(* CoDeSys 2.3.9.35 project: Semaforo3.pro *)
(* Author: Altus *)
(* Libraries: DU35x.lib 7.7.11 15:59:13, Navigation.lib 15.7.11 10:06:00, SysLibTargetVisu.lib 26.11.08 09:53:28, Standard.lib 26.11.08 09:46:20, Iecsfc.lib 26.11.08 09:46:14, SYSLIBCALLBACK.LIB 26.11.08 09:53:30 *)

(* PLC configuration (modules and I/O channels)
Configuração do CP [Root] node -1, in %IB0 out %QB0
  Comunicação [Comunica] node 0, in %IB0 out %QB0
    COM1 [COM1] node 0, in %IB0 out %QB0 {BaudRate = 115200; Paridade = Sem Paridade; StopBits = 1 Stop Bit; Modem = Sem RTS/CTS; Delay = 5}
      MToolIEC [Codesys] node 0, in %IB0 out %QB0
    COM2 [COM2] node 1, in %IB0 out %QB0 {BaudRate = 115200; Paridade = Sem Paridade; StopBits = 1 Stop Bit; Modem = Sem RTS/CTS; Delay = 5}
      Desabilitada [Desabilitado485] node 0, in %IB0 out %QB0
  Barramento [Barramento] node 1, in %IB0 out %QB0
    Entradas [Entradas] node 0, in %IB0 out %QB0
      Entradas Digitais 0 [Entradas0] node 0, in %IW0 out %QB0
        I00 AT %IX0.0 [BitInput] I0.0
        I01 AT %IX0.1 [BitInput] I0.1
        I02 AT %IX0.2 [BitInput] I0.2
        I03 AT %IX0.3 [BitInput] I0.3
        I04 AT %IX0.4 [BitInput] I0.4
        I05 AT %IX0.5 [BitInput] I0.5
        I06 AT %IX0.6 [BitInput] I0.6
        I07 AT %IX0.7 [BitInput] I0.7
        I08 AT %IX0.8 [BitInput] I0.8
      Entradas Digitais 1 [Entradas1] node 0, in %IW1 out %QB0
        I10 AT %IX1.0 [BitInput] I1.0
        I11 AT %IX1.1 [BitInput] I1.1
        I12 AT %IX1.2 [BitInput] I1.2
        I13 AT %IX1.3 [BitInput] I1.3
        I14 AT %IX1.4 [BitInput] I1.4
        I15 AT %IX1.5 [BitInput] I1.5
        I16 AT %IX1.6 [BitInput] I1.6
        I17 AT %IX1.7 [BitInput] I1.7
        I18 AT %IX1.8 [BitInput] I1.8
      Entradas Digitais 2 [Entradas2] node 0, in %IW2 out %QB0
        I20 AT %IX2.0 [BitInput] I2.0
        I21 AT %IX2.1 [BitInput] I2.1
      Entradas Analógicas [EntradaAnalogica] node 0, in %IW4 out %QB0
        AI0 AT %IW4 [WordInput] AI0 {TipoAnalogica = Channel Disable; FiltroAnalogica = Filter 0 - AI=2ms  / AV=90ms; FundoEscala = 0}
        AI1 AT %IW5 [WordInput] AI1 {TipoAnalogica = Channel Disable; FiltroAnalogica = Filter 0 - AI=2ms  / AV=90ms; FundoEscala = 0}
        AI2 AT %IW6 [WordInput] AI2 {TipoAnalogica = Channel Disable; FiltroAnalogica = Filter 0 - AI=2ms  / AV=90ms; FundoEscala = 0}
        AI3 AT %IW7 [WordInput] AI3 {TipoAnalogica = Channel Disable; FiltroAnalogica = Filter 0 - AI=2ms  / AV=90ms; FundoEscala = 0}
      Entradas Rápidas [EntradasRapidas] node 1, in %IB16 out %QB0
        Bloco 0 [Bloco0] node 0, in %IB16 out %QB0
          Desabilitado [DesabilitadoBloco0] node 0, in %IB16 out %QB0
        Bloco 1 [Bloco1] node 1, in %IB16 out %QB0
          Desabilitado [DesabilitadoBloco1] node 0, in %IB16 out %QB0
        Entrada Configuravél Bloco 0 [EntradaConfiBloco0] node 2, in %IB16 out %QB0
          Contador 0 [EntradaConfContador0] node 0, in %IB16 out %QB0 {EntradaConfiguravelContador = Disable}
        Entrada Configuravél Bloco 1 [EntradaConfiBloco1] node 3, in %IB16 out %QB0
          Contador 2 [EntradaConfContador2] node 0, in %IB16 out %QB0 {EntradaConfiguravelContador = Disable}
    Saídas [Saidas] node 1, in %IB13 out %QB0
      Saídas Digitais 0 [Saidas0] node 0, in %IW0 out %QW0
        Q00 AT %QX0.0 [BitOutput] Q0.0
        Q01 AT %QX0.1 [BitOutput] Q0.1
        Q02 AT %QX0.2 [BitOutput] Q0.2
        Q03 AT %QX0.3 [BitOutput] Q0.3
        Q04 AT %QX0.4 [BitOutput] Q0.4
        Q05 AT %QX0.5 [BitOutput] Q0.5
        Q06 AT %QX0.6 [BitOutput] Q0.6
        Q07 AT %QX0.7 [BitOutput] Q0.7
      Saídas Digitais 1 [Saidas1] node 0, in %IW0 out %QW1
        Q10 AT %QX1.0 [BitOutput] Q1.0
        Q11 AT %QX1.1 [BitOutput] Q1.1
        Q12 AT %QX1.2 [BitOutput] Q1.2
        Q13 AT %QX1.3 [BitOutput] Q1.3
        Q14 AT %QX1.4 [BitOutput] Q1.4
        Q15 AT %QX1.5 [BitOutput] Q1.5
        Q16 AT %QX1.6 [BitOutput] Q1.6
        Q17 AT %QX1.7 [BitOutput] Q1.7
      Saídas Analógicas [SaidaAnalogica] node 0, in %IW0 out %QW3
        AO0 AT %QW3 [WordOutput] AO0 {TipoAnalogica = Channel Disable; FundoEscala = 0}
        AO1 AT %QW4 [WordOutput] AO1 {TipoAnalogica = Channel Disable; FundoEscala = 0}
      Saídas Rápidas [SaidasRapidas] node 1, in %IB0 out %QB10
        Saída Rápida 0 Desabilitada [DesabilitadoF0] node 0, in %IB0 out %QB10
        Saída Rápida 1 Desabilitada [DesabilitadoF1] node 1, in %IB0 out %QB10
      Saídas Comum de Contador [SaidasContador] node 2, in %IB0 out %QB10
        Saída do Bloco 0 Desabilitada [DesabilitadoSaidaBloco0] node 0, in %IB0 out %QB10
        Saída do Bloco 1 Desabilitada [DesabilitadoSaidaBloco1] node 1, in %IB0 out %QB10
  Eventos Externos [Eventos] node 2, in %IB13 out %QB6
    Evento Temporizado [TimerEvent] node 0, in %IB13 out %QB6 {Intervalo = 10}
*)

(* Task configuration *)
TASK PRINCIPAL (PRIORITY := 1, INTERVAL := T#1ms);
	PLC_PRG();
END_TASK
TASK NAVIGATION (PRIORITY := 1, INTERVAL := T#20ms);
	NAVEGA();
END_TASK
TASK VISUALIZATION (PRIORITY := 1, INTERVAL := T#500ms);
	MAINTARGETVISU_PAINT_CODE
END_TASK
TASK KEYBOARD_USAGE (PRIORITY := 1, INTERVAL := T#20ms);
	MAINTARGETVISU_INPUT_CODE
END_TASK

(* POU PLC_PRG, LD *)
PROGRAM PLC_PRG

VAR_INPUT
	Ligar AT %IX0.0: BOOL;
	Problema AT %IX0.1: BOOL;
END_VAR
VAR_OUTPUT
	Vermelho AT %QX1.0: BOOL;
	Vermelho2 AT %QX1.1: BOOL;
	Vermelho3 AT %QX1.2: BOOL;
	Vermelho4 AT %QX1.3: BOOL;
	Vermelho5 AT %QX1.4: BOOL;
	Vermelho6 AT %QX1.5: BOOL;
	Verde AT %QX1.7: BOOL;
	Amarelo AT %QX1.6: BOOL;
	Restart: BOOL;
	Pisca: BOOL;
	Vermelhoteste: BOOL;
	VerdeDois: BOOL;
	VermelhoDois: BOOL;
	AmareloDois: BOOL;
END_VAR
VAR
	T1: TON;
	T2: TON;
	T3: TON;
	T4: TON;
	T5: TON;
	T6: TON;
	T7: TON;
	T8: TON;
	Entrada1: INT;
	Tempo_Vermelho: TIME:= T#90s;
	Entrada2: INT;
	Tempo_Amarelo: TIME:= T#4s;
	Entrada3: INT;
	Tempo_Verde: TIME:= T#55s;
	T9: TON;
	Restart2: BOOL;
	T10: TON;
	T11: TON;
END_VAR
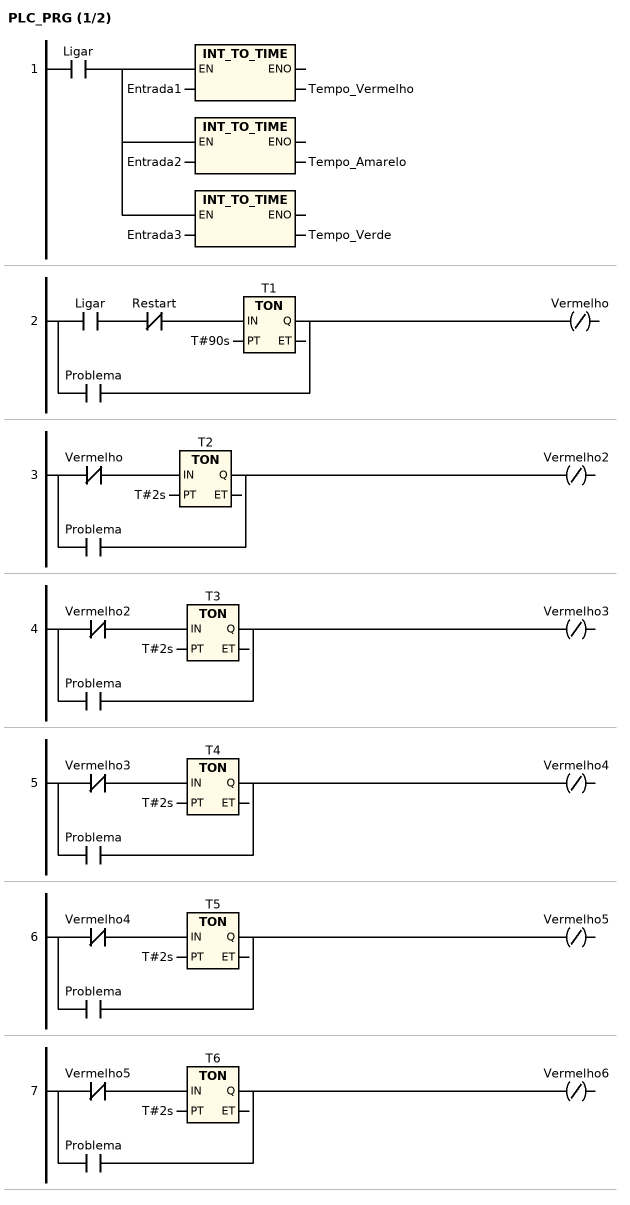
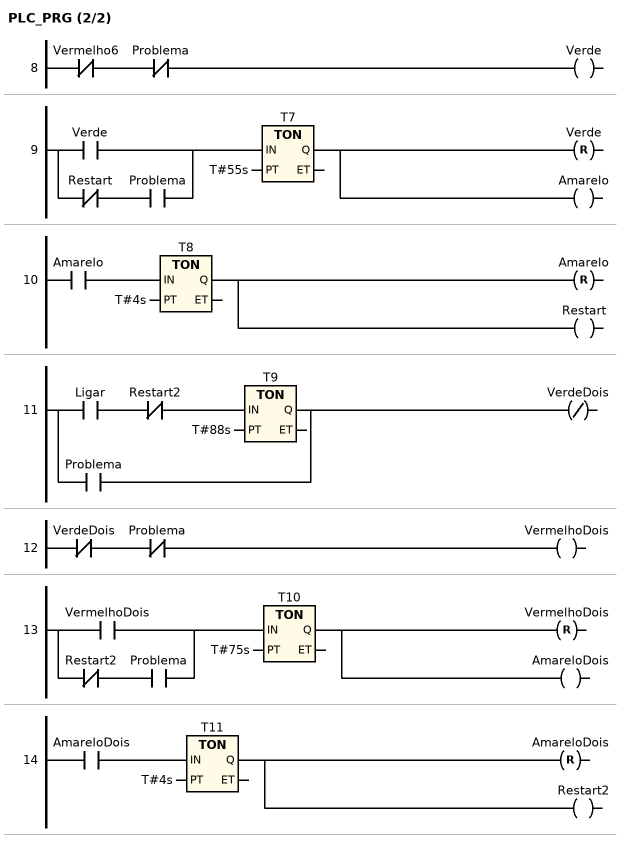
_LD_ (* Ladder Diagram *)
NETWORK 1
	[Ligar]
		EN --- INT_TO_TIME(Entrada1) => Tempo_Vermelho
		EN --- INT_TO_TIME(Entrada2) => Tempo_Amarelo
		EN --- INT_TO_TIME(Entrada3) => Tempo_Verde
NETWORK 2
	{ [Ligar] - [/Restart] - T1:TON(IN: *, PT: T#90s) | [Problema] } --- (/Vermelho)
NETWORK 3
	{ [/Vermelho] - T2:TON(IN: *, PT: T#2s) | [Problema] } --- (/Vermelho2)
NETWORK 4
	{ [/Vermelho2] - T3:TON(IN: *, PT: T#2s) | [Problema] } --- (/Vermelho3)
NETWORK 5
	{ [/Vermelho3] - T4:TON(IN: *, PT: T#2s) | [Problema] } --- (/Vermelho4)
NETWORK 6
	{ [/Vermelho4] - T5:TON(IN: *, PT: T#2s) | [Problema] } --- (/Vermelho5)
NETWORK 7
	{ [/Vermelho5] - T6:TON(IN: *, PT: T#2s) | [Problema] } --- (/Vermelho6)
NETWORK 8
	[/Vermelho6] - [/Problema] --- (Verde)
NETWORK 9
	{ [Verde] | [/Restart] - [Problema] } - T7:TON(IN: *, PT: T#55s) --- (R Verde) (Amarelo)
NETWORK 10
	[Amarelo] - T8:TON(IN: *, PT: T#4s) --- (R Amarelo) (Restart)
NETWORK 11
	{ [Ligar] - [/Restart2] - T9:TON(IN: *, PT: T#88s) | [Problema] } --- (/VerdeDois)
NETWORK 12
	[/VerdeDois] - [/Problema] --- (VermelhoDois)
NETWORK 13
	{ [VermelhoDois] | [/Restart2] - [Problema] } - T10:TON(IN: *, PT: T#75s) --- (R VermelhoDois) (AmareloDois)
NETWORK 14
	[AmareloDois] - T11:TON(IN: *, PT: T#4s) --- (R AmareloDois) (Restart2)
_END_LD_
(* the same logic as Structured Text *)
(* Network 1 *)
IF Ligar THEN
	Tempo_Vermelho := INT_TO_TIME(Entrada1);
	Tempo_Amarelo := INT_TO_TIME(Entrada2);
	Tempo_Verde := INT_TO_TIME(Entrada3);
END_IF;
(* Network 2 *)
T1(IN := Ligar AND NOT Restart, PT := T#90s);
Vermelho := NOT (T1.Q OR Problema);
(* Network 3 *)
T2(IN := NOT Vermelho, PT := T#2s);
Vermelho2 := NOT (T2.Q OR Problema);
(* Network 4 *)
T3(IN := NOT Vermelho2, PT := T#2s);
Vermelho3 := NOT (T3.Q OR Problema);
(* Network 5 *)
T4(IN := NOT Vermelho3, PT := T#2s);
Vermelho4 := NOT (T4.Q OR Problema);
(* Network 6 *)
T5(IN := NOT Vermelho4, PT := T#2s);
Vermelho5 := NOT (T5.Q OR Problema);
(* Network 7 *)
T6(IN := NOT Vermelho5, PT := T#2s);
Vermelho6 := NOT (T6.Q OR Problema);
(* Network 8 *)
Verde := NOT Vermelho6 AND NOT Problema;
(* Network 9 *)
T7(IN := Verde OR NOT Restart AND Problema, PT := T#55s);
IF T7.Q THEN Verde := FALSE; END_IF;
Amarelo := T7.Q;
(* Network 10 *)
T8(IN := Amarelo, PT := T#4s);
IF T8.Q THEN Amarelo := FALSE; END_IF;
Restart := T8.Q;
(* Network 11 *)
T9(IN := Ligar AND NOT Restart2, PT := T#88s);
VerdeDois := NOT (T9.Q OR Problema);
(* Network 12 *)
VermelhoDois := NOT VerdeDois AND NOT Problema;
(* Network 13 *)
T10(IN := VermelhoDois OR NOT Restart2 AND Problema, PT := T#75s);
IF T10.Q THEN VermelhoDois := FALSE; END_IF;
AmareloDois := T10.Q;
(* Network 14 *)
T11(IN := AmareloDois, PT := T#4s);
IF T11.Q THEN AmareloDois := FALSE; END_IF;
Restart2 := T11.Q;
END_PROGRAM

(* POU NAVEGA, ST *)
PROGRAM NAVEGA
VAR
	ControleTelas : NAVIGATION;
	ListaTelas 	: ARRAY [0..30] OF STRING(10);
END_VAR
(* Adiciona a tela MAIN como tela principal *)
ListaTelas[0] := 'MAIN';

(* Ativa o controle automático de navegação somente pelo teclado *)
ControleTelas(ENABLE_UPDW := FALSE, VISU_LIST := ListaTelas, UP := FALSE , DOWN := FALSE);
END_PROGRAM

(* Visualisation MAIN
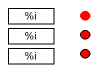
rectangle at (14,6)-(60,22): text "%i"; shows PLC_PRG.Entrada1; editable 2..300000
rectangle at (14,26)-(60,42): text "%i"; shows PLC_PRG.Entrada2; editable 2..300000
rectangle at (14,46)-(60,62): text "%i"; shows PLC_PRG.Entrada3; editable 2..300000
ellipse at (86,9)-(96,18): alarm colour if PLC_PRG.VermelhoDois
ellipse at (86,28)-(96,37): alarm colour if PLC_PRG.AmareloDois
ellipse at (86,47)-(96,56): alarm colour if PLC_PRG.VerdeDois
*)
